// TwinCAT 3 PLC project main
// ProgramVersion: 3.1.4024.0
// libraries:
//   Tc2_Standard, * (Beckhoff Automation GmbH)
//   Tc2_System, * (Beckhoff Automation GmbH)
//   Tc3_Module, * (Beckhoff Automation GmbH)
// project tree:
//   DUTs/ PID_Parameter_Strukt.TcDUT, PT1T2_Parameter_Strukt.TcDUT, System_Modus_Enum.TcDUT
//   / PlcTask.TcTTO
//   POUs/ MAIN.TcPOU, PID_Regler.TcPOU, PT1T2_Prozess.TcPOU
// real-time tasks:
//   TASK PlcTask: cycle T#10ms, priority 20, ADS port 350

CONFIGURATION main
    RESOURCE PLC ON TwinCAT3
        TASK PlcTask(INTERVAL := T#10ms, PRIORITY := 20);
        PROGRAM MAIN WITH PlcTask : MAIN;
    END_RESOURCE
END_CONFIGURATION

// ---- DUTs/PID_Parameter_Strukt.TcDUT
TYPE PID_Parameter_Strukt :
STRUCT
	Kp :		REAL;
	Ti :		REAL;
	Td :		REAL;
	N :			REAL;
	ARW :		REAL;
	umin :		REAL;
	umax :		REAL;
END_STRUCT
END_TYPE

// ---- DUTs/PT1T2_Parameter_Strukt.TcDUT
TYPE PT1T2_Parameter_Strukt :
STRUCT
	K :			REAL;
	T1 :		REAL;
	T2 :		REAL;
END_STRUCT
END_TYPE

// ---- DUTs/System_Modus_Enum.TcDUT
{attribute 'qualified_only'}
{attribute 'strict'}
TYPE System_Modus_Enum :
(
	System_Init := 0,
	System_Run
);
END_TYPE

// ---- POUs/MAIN.TcPOU
PROGRAM MAIN
VAR
END_VAR

END_PROGRAM

// ---- POUs/PID_Regler.TcPOU
FUNCTION_BLOCK PID_Regler
VAR_INPUT
	R :			REAL;
	Y :			REAL;
	Modus :		System_Modus_Enum;
	Param :		PID_Parameter_Strukt;
	T :			REAL;
END_VAR
VAR_OUTPUT
END_VAR
VAR
END_VAR

CASE Modus OF
	System_Modus_Enum.System_Init:
	;
	System_Modus_Enum.System_Run:
	;
END_CASE

END_FUNCTION_BLOCK

// ---- POUs/PT1T2_Prozess.TcPOU
FUNCTION_BLOCK PT1T2_Prozess
VAR_INPUT
	u :			REAL;
	Modus :		System_Modus_Enum;
	Param :		PT1T2_Parameter_Strukt;
	T :			REAL;
END_VAR
VAR_OUTPUT
	y :			REAL;
END_VAR
VAR
	a1 :		REAL;
	a2 :		REAL;
	b0 :		REAL;
	b1 :		REAL;
	b2 :		REAL;
	
	ym :		REAL;
	ymm :		REAL;
END_VAR

CASE Modus OF
	System_Modus_Enum.System_Init:
	a1 := T + Param.T1;
	a2 := T + Param.T2;
	b0 := (Param.K*T*T)/(a1*a2);
	b1 := -(Param.T1/a1+Param.T2/a2);
	b2 := (Param.T1*Param.T2)/(a1*a2);
	ym := 0;
	ymm := 0;
	;
	System_Modus_Enum.System_Run:
	y := -a1 * ym - a2 *ymm + b0 * u;
	ym := y;
	ymm := ym;
	;
END_CASE

END_FUNCTION_BLOCK
